_CFC_ (* Continuous Function Chart, elements in execution order *)
#0 ABS(SCHU_P2_1_YA4_RASSOG)
#1 GT(#0, SCHU_P2_1_YA4_UST_RAS_TEMP)
#2 AND(SCHU_P2_1_UST_RE_RABOTA, #1)
#3 INT_TO_TIME(SCHU_P2_1_YA4_ZADER_OTK_TEMP)
#4 MUL(#3, 1000)
#5 YA4_ZADER_TEMP:TON(IN: #2, PT: #4)
#6 ABS(SCHU_P2_1_YA4_RASSOG_POL)
#7 GT(#6, SCHU_P2_1_YA4_UST_RAS_POL)
#8 AND(SCHU_P2_1_UST_RE_RABOTA, #7)
#9 INT_TO_TIME(SCHU_P2_1_YA4_ZADER_OTK)
#10 MUL(#9, 1000)
#11 YA4_ZADER_POL:TON(IN: #8, PT: #10)
#12 OR(#5.Q, #11.Q)
#13 AND(SCHU_P2_1_UE3_T_DOST, SCHU_P2_1_SA6_DI7_A, #12)
#14 RS_YA4_OTKZ:SR(SET1: #13, RESET: SCHU_P2_1_SB)
#15 SCHU_P2_1_Z_YA4_OTKAZ <= #14.Q1
_END_CFC_
(* the same logic as Structured Text *)
YA4_ZADER_TEMP(IN := SCHU_P2_1_UST_RE_RABOTA AND (ABS(SCHU_P2_1_YA4_RASSOG) > SCHU_P2_1_YA4_UST_RAS_TEMP), PT := INT_TO_TIME(SCHU_P2_1_YA4_ZADER_OTK_TEMP) * 1000);
YA4_ZADER_POL(IN := SCHU_P2_1_UST_RE_RABOTA AND (ABS(SCHU_P2_1_YA4_RASSOG_POL) > SCHU_P2_1_YA4_UST_RAS_POL), PT := INT_TO_TIME(SCHU_P2_1_YA4_ZADER_OTK) * 1000);
RS_YA4_OTKZ(SET1 := SCHU_P2_1_UE3_T_DOST AND SCHU_P2_1_SA6_DI7_A AND (YA4_ZADER_TEMP.Q OR YA4_ZADER_POL.Q), RESET := SCHU_P2_1_SB);
SCHU_P2_1_Z_YA4_OTKAZ := RS_YA4_OTKZ.Q1;
END_PROGRAM

(* POU TZBiS/TZB/Z_Zam, CFC *)
PROGRAM Z_Zam
VAR
	RT_VKL: R_TRIG;
	SR_ZAM: SR;
	TON_VKL: TON;
	TP_VKL: TON;
	FT_TP_VKL: F_TRIG;
	SR_TS: SR;
END_VAR
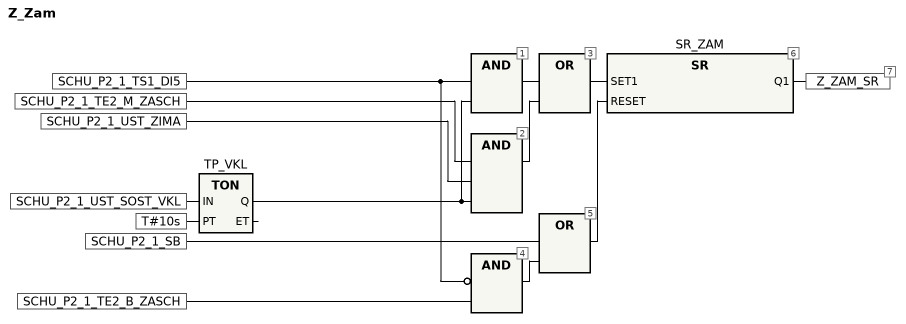
_CFC_ (* Continuous Function Chart, elements in execution order *)
#0 TP_VKL:TON(IN: SCHU_P2_1_UST_SOST_VKL, PT: T#10s)
#1 AND(SCHU_P2_1_TS1_DI5, #0.Q)
#2 AND(SCHU_P2_1_TE2_M_ZASCH, SCHU_P2_1_UST_ZIMA, #0.Q)
#3 OR(#1, #2)
#4 AND(NOT SCHU_P2_1_TS1_DI5, SCHU_P2_1_TE2_B_ZASCH)
#5 OR(SCHU_P2_1_SB, #4)
#6 SR_ZAM:SR(SET1: #3, RESET: #5)
#7 Z_ZAM_SR <= #6.Q1
_END_CFC_
(* the same logic as Structured Text *)
TP_VKL(IN := SCHU_P2_1_UST_SOST_VKL, PT := T#10s);
SR_ZAM(SET1 := (SCHU_P2_1_TS1_DI5 AND TP_VKL.Q) OR (SCHU_P2_1_TE2_M_ZASCH AND SCHU_P2_1_UST_ZIMA AND TP_VKL.Q), RESET := SCHU_P2_1_SB OR (NOT SCHU_P2_1_TS1_DI5 AND SCHU_P2_1_TE2_B_ZASCH));
Z_ZAM_SR := SR_ZAM.Q1;
END_PROGRAM

(* POU TZBiS/TZB/Z_Dlit_Ster_Reg, CFC *)
	PROGRAM Z_Dlit_Ster_Reg
VAR
	SR_HZ20S60: SR;
	LT_HZm20: ISTOK_LT;
	TON_HZm20: TON;
END_VAR
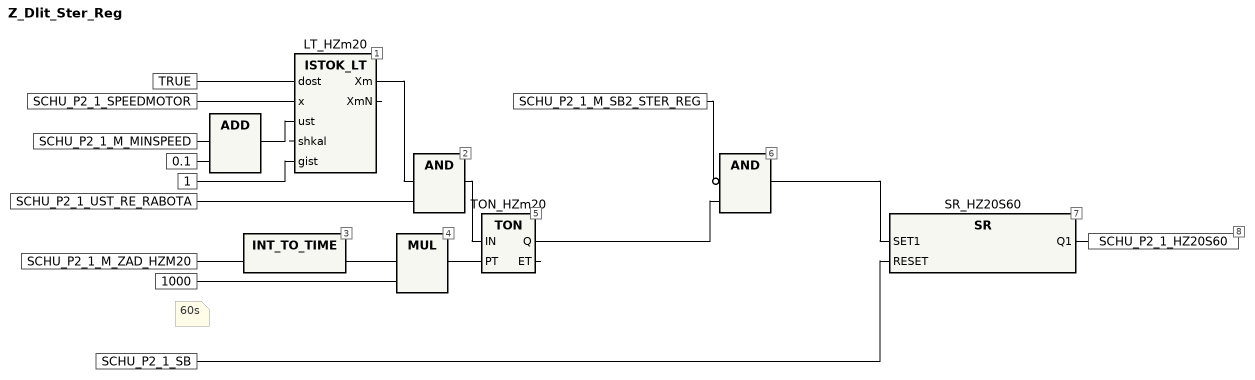
_CFC_ (* Continuous Function Chart, elements in execution order *)
(* 60s *)
#0 ADD(SCHU_P2_1_M_MINSPEED, 0.1)
#1 LT_HZm20:ISTOK_LT(dost: TRUE, x: SCHU_P2_1_SPEEDMOTOR, ust: #0, shkal: -, gist: 1)
#2 AND(#1.Xm, SCHU_P2_1_UST_RE_RABOTA)
#3 INT_TO_TIME(SCHU_P2_1_M_ZAD_HZM20)
#4 MUL(#3, 1000)
#5 TON_HZm20:TON(IN: #2, PT: #4)
#6 AND(NOT SCHU_P2_1_M_SB2_STER_REG, #5.Q)
#7 SR_HZ20S60:SR(SET1: #6, RESET: SCHU_P2_1_SB)
#8 SCHU_P2_1_HZ20S60 <= #7.Q1
_END_CFC_
(* the same logic as Structured Text *)
(* 60s *)
LT_HZm20(dost := TRUE, x := SCHU_P2_1_SPEEDMOTOR, ust := SCHU_P2_1_M_MINSPEED + 0.1, gist := 1);
TON_HZm20(IN := LT_HZm20.Xm AND SCHU_P2_1_UST_RE_RABOTA, PT := INT_TO_TIME(SCHU_P2_1_M_ZAD_HZM20) * 1000);
SR_HZ20S60(SET1 := NOT SCHU_P2_1_M_SB2_STER_REG AND TON_HZm20.Q, RESET := SCHU_P2_1_SB);
SCHU_P2_1_HZ20S60 := SR_HZ20S60.Q1;
END_PROGRAM

(* POU TZBiS/TZB/Z_ALL, CFC *)
PROGRAM Z_ALL
VAR
	SR_Z_all: SR;
END_VAR
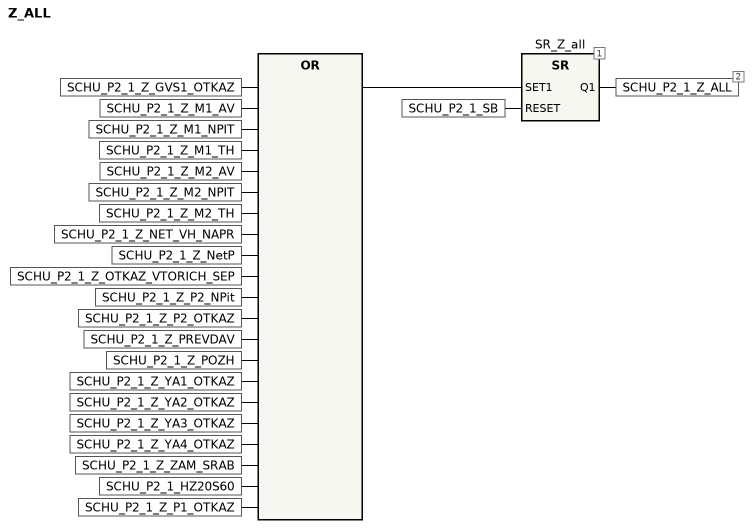
_CFC_ (* Continuous Function Chart, elements in execution order *)
#0 OR(SCHU_P2_1_Z_GVS1_OTKAZ, SCHU_P2_1_Z_M1_AV, SCHU_P2_1_Z_M1_NPIT, SCHU_P2_1_Z_M1_TH, SCHU_P2_1_Z_M2_AV, SCHU_P2_1_Z_M2_NPIT, SCHU_P2_1_Z_M2_TH, SCHU_P2_1_Z_NET_VH_NAPR, SCHU_P2_1_Z_NetP, SCHU_P2_1_Z_OTKAZ_VTORICH_SEP, SCHU_P2_1_Z_P2_NPit, SCHU_P2_1_Z_P2_OTKAZ, SCHU_P2_1_Z_PREVDAV, SCHU_P2_1_Z_POZH, SCHU_P2_1_Z_YA1_OTKAZ, SCHU_P2_1_Z_YA2_OTKAZ, SCHU_P2_1_Z_YA3_OTKAZ, SCHU_P2_1_Z_YA4_OTKAZ, SCHU_P2_1_Z_ZAM_SRAB, SCHU_P2_1_HZ20S60, SCHU_P2_1_Z_P1_OTKAZ)
#1 SR_Z_all:SR(SET1: #0, RESET: SCHU_P2_1_SB)
#2 SCHU_P2_1_Z_ALL <= #1.Q1
_END_CFC_
(* the same logic as Structured Text *)
SR_Z_all(SET1 := SCHU_P2_1_Z_GVS1_OTKAZ OR SCHU_P2_1_Z_M1_AV OR SCHU_P2_1_Z_M1_NPIT OR SCHU_P2_1_Z_M1_TH OR SCHU_P2_1_Z_M2_AV OR SCHU_P2_1_Z_M2_NPIT OR SCHU_P2_1_Z_M2_TH OR SCHU_P2_1_Z_NET_VH_NAPR OR SCHU_P2_1_Z_NetP OR SCHU_P2_1_Z_OTKAZ_VTORICH_SEP OR SCHU_P2_1_Z_P2_NPit OR SCHU_P2_1_Z_P2_OTKAZ OR SCHU_P2_1_Z_PREVDAV OR SCHU_P2_1_Z_POZH OR SCHU_P2_1_Z_YA1_OTKAZ OR SCHU_P2_1_Z_YA2_OTKAZ OR SCHU_P2_1_Z_YA3_OTKAZ OR SCHU_P2_1_Z_YA4_OTKAZ OR SCHU_P2_1_Z_ZAM_SRAB OR SCHU_P2_1_HZ20S60 OR SCHU_P2_1_Z_P1_OTKAZ, RESET := SCHU_P2_1_SB);
SCHU_P2_1_Z_ALL := SR_Z_all.Q1;
END_PROGRAM

(* POU Regim/ALL_Regim, CFC *)
PROGRAM ALL_Regim
VAR
END_VAR
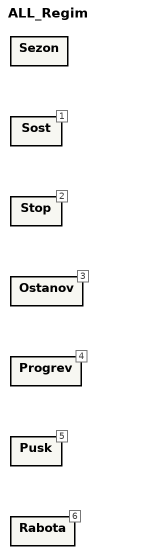
_CFC_ (* Continuous Function Chart, elements in execution order *)
#0 Sezon()
#1 Sost()
#2 Stop()
#3 Ostanov()
#4 Progrev()
#5 Pusk()
#6 Rabota()
_END_CFC_
(* the same logic as Structured Text *)
Sezon();
Sost();
Stop();
Ostanov();
Progrev();
Pusk();
Rabota();
END_PROGRAM

(* POU Regim/Sezon, CFC *)
PROGRAM Sezon
VAR
	RS_Sezon: RS;
	RT_Zima: R_TRIG;
	RT_Leto: R_TRIG;
	RT_Auto: R_TRIG;
	RS_Auto: RS;
	RT_T: R_TRIG;
END_VAR
VAR (* helpers for the ST form of the networks *)
	_t72 : BOOL;
END_VAR
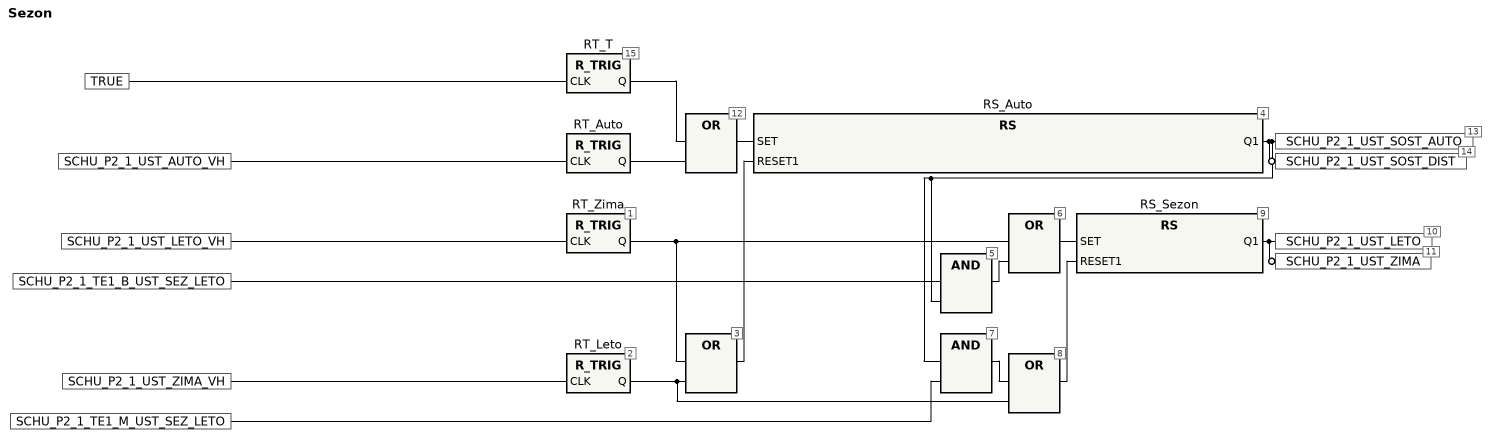
_CFC_ (* Continuous Function Chart, elements in execution order *)
#0 RT_Auto:R_TRIG(CLK: SCHU_P2_1_UST_AUTO_VH)
#1 RT_Zima:R_TRIG(CLK: SCHU_P2_1_UST_LETO_VH)
#2 RT_Leto:R_TRIG(CLK: SCHU_P2_1_UST_ZIMA_VH)
#3 OR(#1.Q, #2.Q)
#4 RS_Auto:RS(SET: #12, RESET1: #3)
#5 AND(SCHU_P2_1_TE1_B_UST_SEZ_LETO, #4.Q1)
#6 OR(#1.Q, #5)
#7 AND(#4.Q1, SCHU_P2_1_TE1_M_UST_SEZ_LETO)
#8 OR(#7, #2.Q)
#9 RS_Sezon:RS(SET: #6, RESET1: #8)
#10 SCHU_P2_1_UST_LETO <= #9.Q1
#11 SCHU_P2_1_UST_ZIMA <= NOT #9.Q1
#12 OR(#15.Q, #0.Q)
#13 SCHU_P2_1_UST_SOST_AUTO <= #4.Q1
#14 SCHU_P2_1_UST_SOST_DIST <= NOT #4.Q1
#15 RT_T:R_TRIG(CLK: TRUE)
_END_CFC_
(* the same logic as Structured Text *)
RT_Auto(CLK := SCHU_P2_1_UST_AUTO_VH);
RT_Zima(CLK := SCHU_P2_1_UST_LETO_VH);
RT_Leto(CLK := SCHU_P2_1_UST_ZIMA_VH);
RS_Auto(SET := _t72, RESET1 := RT_Zima.Q OR RT_Leto.Q);
RS_Sezon(SET := RT_Zima.Q OR (SCHU_P2_1_TE1_B_UST_SEZ_LETO AND RS_Auto.Q1), RESET1 := (RS_Auto.Q1 AND SCHU_P2_1_TE1_M_UST_SEZ_LETO) OR RT_Leto.Q);
SCHU_P2_1_UST_LETO := RS_Sezon.Q1;
SCHU_P2_1_UST_ZIMA := NOT RS_Sezon.Q1;
_t72 := RT_T.Q OR RT_Auto.Q;
SCHU_P2_1_UST_SOST_AUTO := RS_Auto.Q1;
SCHU_P2_1_UST_SOST_DIST := NOT RS_Auto.Q1;
RT_T(CLK := TRUE);
END_PROGRAM

(* POU Regim/Sost, CFC *)
PROGRAM Sost
VAR
	RS_Sost: RS;
	RT_PUSK: R_TRIG;
	RT_STOP: R_TRIG;
	RS_Old_Sost: RS;
	TON_Kv1: TON;
	TON_Kv1_1: TON;
	OLD_SOST: BOOL;

	KV1: BOOL;
	RT_PUSK_OLD: R_TRIG;
	CTU_TS: CTU;
	TOF_TS_1: TOF;
	TOF_TS_2: TOF;
	TOF_TS_3: TOF;
	RT_PUSK_OLD1: R_TRIG;
	TON_Kv1_11: TON;
	TON_Kv11: TON;
	TOF_TE_1: TOF;
	TOF_Te_2: TOF;
	TOF_Te_3: TOF;
	CTU_Te: CTU;
END_VAR
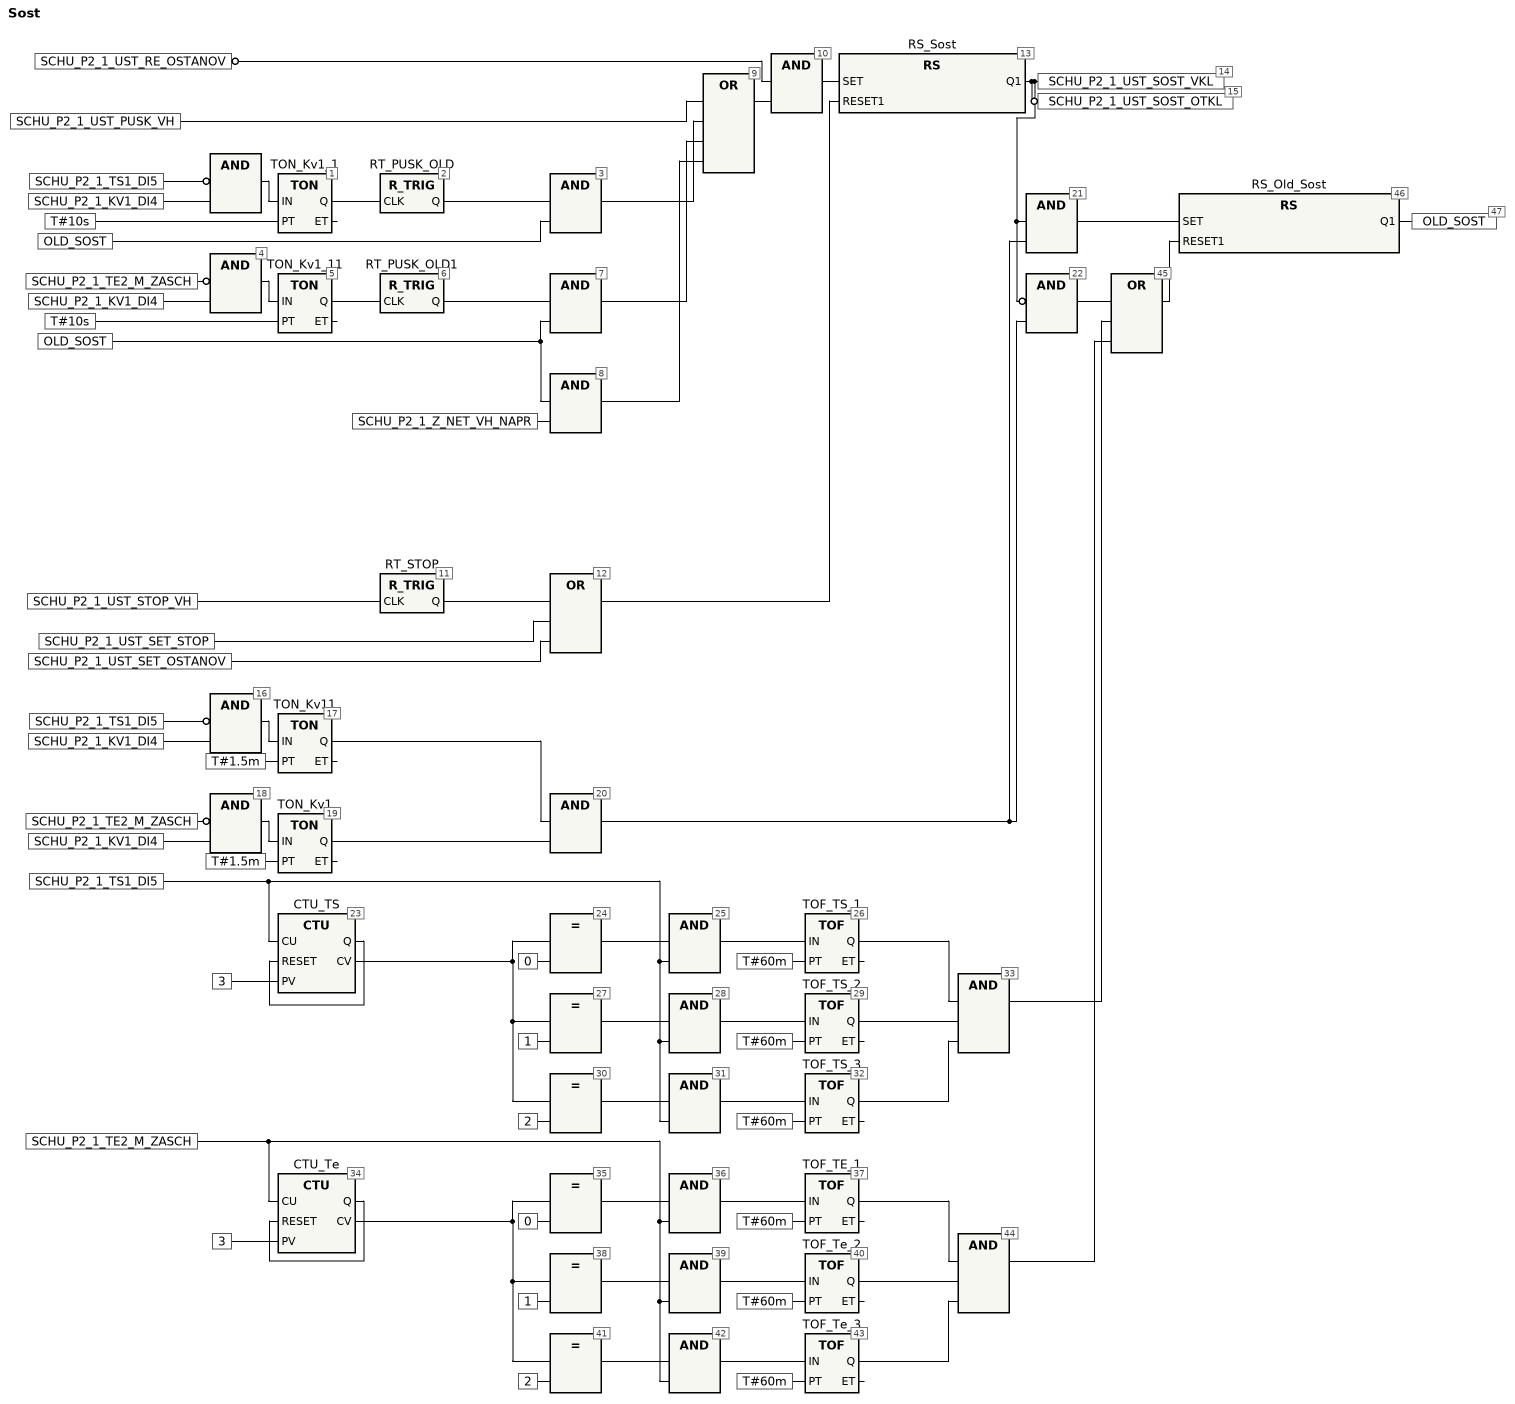
